FUNCTION_BLOCK FB_HMI_SP_Alarm
VAR_INPUT
	Error						: BOOL;
	ErrorID						: DINT;
	aAlarm						: POINTER TO FB_TcAlarm;
	wAlarm						: POINTER TO DWORD;
	SourceName					: STRING;
	TcSourceInfo				: FB_TcSourceInfo;
	TcEventLogger 				: FB_TcEventLogger;
	EventId						: UDINT;
END_VAR
VAR
	bResult : BOOL;
	AlarmExist						: ARRAY[0..G.MAX_ALR] OF BOOL;
END_VAR

bResult := FALSE;
IF Error THEN
	CASE ErrorID OF
		1010://Execute error
			wAlarm^.2 := 1;
			
			IF NOT AlarmExist[2] THEN 
				AlarmExist[2] := TRUE; 
				bResult := FC_AlarmExists(SourceName, TcSourceInfo, TcEventLogger, aAlarm[2], TC_Events.DB_Alarm.A50102, (EventId + 2));
			ELSE 
				bResult := TRUE; 
			END_IF
			
			IF bResult THEN
				aAlarm[2].Raise(0);
			END_IF
		1020://read error
			wAlarm^.3 := 1;
			
			IF NOT AlarmExist[3] THEN 
				AlarmExist[3] := TRUE; 
				bResult := FC_AlarmExists(SourceName, TcSourceInfo, TcEventLogger, aAlarm[3], TC_Events.DB_Alarm.A50103, (EventId + 3));
			ELSE 
				bResult := TRUE; 
			END_IF
			IF bResult THEN
				aAlarm[3].Raise(0);	
			END_IF
		1999://Timeout
			wAlarm^.1 := 1;
			
			IF NOT AlarmExist[1] THEN 
				AlarmExist[1] := TRUE; 
				bResult := FC_AlarmExists(SourceName, TcSourceInfo, TcEventLogger, aAlarm[1], TC_Events.DB_Alarm.A50101, (EventId + 1));
			ELSE 
				bResult := TRUE; 
			END_IF
			IF bResult THEN
				aAlarm[1].Raise(0);
			END_IF
		ELSE // Generic
			wAlarm^.0 := 1;
			
			IF NOT AlarmExist[0] THEN 
				AlarmExist[0] := TRUE; 
				bResult := FC_AlarmExists(SourceName, TcSourceInfo, TcEventLogger, aAlarm[0], TC_Events.DB_Alarm.A50100, (EventId + 0));
			ELSE 
				bResult := TRUE; 
			END_IF
			IF bResult THEN
				aAlarm[0].ipArguments.Clear().AddDInt(ErrorID);
				aAlarm[0].Raise(0);	
			END_IF
	END_CASE
END_IF

END_FUNCTION_BLOCK

(* stored: Version 1.1.0.1, ProductVersion 3.1.4024.15
   POU FB_HMI_SP_Alarm: Id {a3e4b17a-19cc-41cb-9f79-0e5893d7606a}, SpecialFunc None *)
